Staubli VAL3: onF6Event.pgx

program onF6Event()
  local string l_sItem
  local string l_sPage
begin
  // look if the bButton is enable
  if bButton[5]
    //
    //
    l_sPage="kernel/page/frame"
    call loadPage(l_sPage,l_sItem)
    logMsg("[KERNEL] INTERFACE:PAGE Home Page")
  endIf
end
